FUNCTION_BLOCK AX_TP (* standard timer function block (pulse) *)
  (* Standard: 61499-2; Classification: standard timer function block; Description: Copyright (c) 2024 HR Agrartechnik GmbH This program and the accompanying materials are made available under the terms of the Eclipse Public License 2.0 which is available at https://www.eclipse.org/legal/epl-2.0/ SPDX-License-Identifier: EPL-2.0 *)
  (* Version 3.0, 2025-04-14, Patrick Aigner, changed package *)
  (* Version 1.1, 2024-04-23, Franz Hoepfinger, HR Agrartechnik GmbH, Add a Reset to Timer FBs *)
  (* Version 1.0, 2024-03-04, Franz Hoepfinger, HR Agrartechnik GmbH *)
  PACKAGE adapter::events::unidirectional::timers;
  IMPORT eclipse4diac::core::TypeHash;
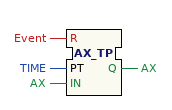
  EVENT_INPUT
    R; (* Reset *)
  END_EVENT
  VAR_INPUT
    PT : TIME; (* Pulse time *)
  END_VAR
  SOCKETS
    IN : adapter::types::unidirectional::AX; (* Input *)
  END_SOCKETS
  PLUGS
    Q : adapter::types::unidirectional::AX; (* Output *)
  END_PLUGS
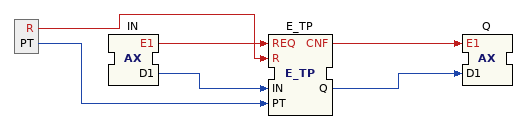
  FBS
    E_TP : iec61499::events::timers::E_TP;
  END_FBS
  EVENT_CONNECTIONS
    IN.E1 TO E_TP.REQ;
    R TO E_TP.R;
    E_TP.CNF TO Q.E1;
  END_CONNECTIONS
  DATA_CONNECTIONS
    IN.D1 TO E_TP.IN;
    PT TO E_TP.PT;
    E_TP.Q TO Q.D1;
  END_CONNECTIONS
END_FUNCTION_BLOCK
